(* PLC project EPEC_CU2.project, CODESYS V3.5 SP19, author XXXX *)
(* stored: creationDateTime 2026-03-19T14:01:24.5182463+02:00, modificationDateTime 2026-03-19T14:01:24.5182463+02:00, organization XXXX *)

{attribute 'analysis' := '-16, -33'}
TYPE FastParameters : STRUCT
  FastParameter1 : BYTE;
  FastParameter2 : WORD;
  FastParameter3 : DWORD;
END_STRUCT;
END_TYPE

(* This PRG contains non safety-related code. The following attribute is autogenerated. Do not remove. *)
{attribute 'location' := '16#800'}
PROGRAM Main

                    ;

                  
END_PROGRAM

(* This PRG contains non safety-related code. The following attribute is autogenerated. Do not remove. *)
{attribute 'location' := '16#800'}
PROGRAM MainInit
  VAR_OUTPUT
    o_MainInitReady : BOOL := FALSE;
  END_VAR

                    o_MainInitReady := TRUE;
                  
END_PROGRAM

PROGRAM S_Main

                    
(*
  Following features are application controlled using product specific HW diagnostic program:
  - Safety switch startup test
  - Safety switch (output group 1) control
  
  Following example can be used for controlling. Add application specific conditions.
*)
// Safety switch startup test trigger. Add a system specific delay if necessary.
// For example, if there are voltage fluctuations during system startup.
EPEC_HWDIAG.S_CORE1MCU_Diagnostic.i_SwitchStartupTestEnable := TRUE;

// Safety switch control
EPEC_HWDIAG.S_CORE1MCU_Diagnostic.i_OutputGroup1Control := G_StatusFlags_Safe.S_SafeOperationEnable;

(* HW diagnostic program contains supply voltage states for different control types which are used by application
  Example:
	output1 := control AND // application control
				G_StatusFlags_Safe.S_SafeOperationEnable AND // common diagnostic OK conditions
				EPEC_HWDIAG.S_CORE1MCU_Diagnostic.o_SupplyVoltageEnableStates.SafeControl; // supply voltage in safe control operational range
*)

// For more information, see Epec programming manual's How to guides.									
										
                  
END_PROGRAM

PROGRAM S_MainInit
  VAR_OUTPUT
    o_MainInitReady : BOOL := FALSE;
  END_VAR

                    o_MainInitReady := TRUE;

                  
END_PROGRAM

(* NOTE! NOTE! NOTE! NOTE! NOTE! NOTE! NOTE! NOTE! NOTE! NOTE! NOTE! This object is created by Epec MultiTool User changes are overwritten when project is imported Content(input conversion, validation and diagnostic): - Validate all safe inputs using * S_ADCToVoltageOrCurrent() * S_ValidateAI() * S_VoltageToDI() * S_ValidateDI() * S_AIOverCurrentProtection(). All FB's o_Status.OutputValid output statuses will be taken in count into 'inputs valid' status. This PRG contains safety-related code. The following attribute is autogenerated. Do not remove. *)
{attribute 'hide_all_locals'}
{attribute 'analysis' := '-3, -9, -29, -33, -35, -130'}
PROGRAM S_Inputs
  VAR_INPUT
    i_Enable : BOOL := TRUE;
    i_Initialize : BOOL := TRUE;
  END_VAR
  VAR_OUTPUT
    o_InitReady : BOOL := FALSE;
    o_AI_VIN_V_Diagnostic : DWORD;  (* Filtered ADC value for supply voltage (VIN_M) *)
    o_AI_PCB_1_V_Diagnostic : DWORD;  (* Filtered ADC value for PCB1 temperature *)
    o_AI_PCB_2_V_Diagnostic : DWORD;  (* Filtered ADC value for PCB2 temperature *)
    o_AI_MCU_C_Diagnostic : DINT;  (* MCU temperature [0.1 C] *)
    o_AI_SBC_C_Diagnostic : DINT;  (* SBC temperature [0.1 C] *)
    o_AI_VOUT_SAFE_Diagnostic : DWORD;  (* Filtered ADC value for voltage after safety switch (VOUT_SAFE_M) *)
    o_AI_VOUT_NON_SAFE_Diagnostic : DWORD;  (* Filtered ADC value for voltage before safety switch (VOUT_NONSAFE_M) *)
    o_AI_BSL_V_Diagnostic : DWORD;  (* Filtered ADC value for BSL voltage *)
    o_DI_FACTORY_RESET_Diagnostic : BYTE;  (* Factory reset state *)
    o_DI_SERVICE_MODE_Diagnostic : BYTE;  (* Service mode state *)
    o_UptimeWarning_Diagnostic : BOOL;  (* Uptime warning, maximum runtime approaching *)
    o_UptimeExceeded_Diagnostic : BOOL;  (* Uptime exceeded, runtime after bootup over limit *)
    o_Uptime_Elapsed_Diagnostic : TIME;  (* Elapsed time since bootup, counts up to the allowed 24h *)
  END_VAR
  VAR
    AI_VIN_V_Diagnostic : DWORD;  (* Internal diagnostic variable mapped to FW io interface *)
    AI_PCB_1_V_Diagnostic : DWORD;  (* Internal diagnostic variable mapped to FW io interface *)
    AI_PCB_2_V_Diagnostic : DWORD;  (* Internal diagnostic variable mapped to FW io interface *)
    AI_MCU_C_Diagnostic : DINT;  (* Internal diagnostic variable mapped to FW io interface *)
    AI_SBC_C_Diagnostic : DINT;  (* Internal diagnostic variable mapped to FW io interface *)
    AI_VOUT_SAFE_Diagnostic : DWORD;  (* Internal diagnostic variable mapped to FW io interface *)
    AI_VOUT_NON_SAFE_Diagnostic : DWORD;  (* Internal diagnostic variable mapped to FW io interface *)
    AI_BSL_V_Diagnostic : DWORD;  (* Internal diagnostic variable mapped to FW io interface *)
    DI_FACTORY_RESET_Diagnostic : BYTE;  (* Internal diagnostic variable mapped to FW io interface *)
    DI_SERVICE_MODE_Diagnostic : BYTE;  (* Internal diagnostic variable mapped to FW io interface *)
    uptimeWarningTimer_Diagnostic : Standard.TON;  (* TON timer for uptime warning *)
    uptimeExceededTimer_Diagnostic : Standard.TON;  (* TON timer for uptime exceeded *)
  END_VAR

                    IF(i_Initialize) THEN
	o_InitReady:= TRUE;
¤#INIT_S_INPUTS_INIT#¤  
ELSE
¤#INIT_S_INPUTS_CODE#¤  
END_IF

                  
END_PROGRAM

(* NOTE! NOTE! NOTE! NOTE! NOTE! NOTE! NOTE! NOTE! NOTE! NOTE! NOTE! This object is created by Epec MultiTool User changes are overwritten when project is imported Content - Init and update all used SafeSSeriesDiagnostic library FB instances * S_DOControlAndDiagnostics() * S_DOValveEcoControlAndDiagnostics() All Init methods return TRUE if ok. They will be taken in count into Ready status. This PRG contains non safety-related code. The following attribute is autogenerated. Do not remove. *)
{attribute 'hide_all_locals'}
{attribute 'analysis' := '-3, -9, -29, -33, -35, -130'}
PROGRAM S_Outputs
  VAR_INPUT
    i_Enable : BOOL := TRUE;
    i_Initialize : BOOL := TRUE;
    i_UpdateMeasurements : BOOL := FALSE;
  END_VAR
  VAR_OUTPUT
    o_InitReady : BOOL := FALSE;
    o_TotalOutputCurrent_Diagnostic : DINT;  (* Sum of all output current measurements *)
  END_VAR
  VAR
    TotalOutputCurrent_Diagnostic : DINT;  (* Sum of all output current measurements *)
    pin : DWORD := DWORD#0;
    connector : DWORD := DWORD#0;
    info1 : DWORD := DWORD#0;
    info2 : DWORD := DWORD#0;
    errorCode : DINT := DINT#0;
  END_VAR

                    IF(i_Initialize) THEN
	o_InitReady:= TRUE;
¤#INIT_S_OUTPUTS_INIT#¤  
ELSIF i_UpdateMeasurements THEN
¤#S_OUTPUTS_MEASUREMENT#¤  
;
ELSE
¤#INIT_S_OUTPUTS_CODE#¤  
END_IF

                  
END_PROGRAM

CONFIGURATION Device
  RESOURCE Application ON PLC
    TASK NonSafePRG_TASK(INTERVAL := T#10ms, PRIORITY := 1);
    TASK SafePRG_TASK(INTERVAL := T#10ms, PRIORITY := 0);
    PROGRAM PLC_PRG WITH NonSafePRG_TASK : PLC_PRG;
    PROGRAM S_PLC_PRG WITH SafePRG_TASK : S_PLC_PRG;
  END_RESOURCE
END_CONFIGURATION
